# EPICS IOC start-up script: iocsh/streamMail.iocsh
################################################################################
#
# streamMail.iocsh
#
# Loads 10 user Notifiers
#
# PREFIX	- PV prefix
# MSERVER 	- mail server
# ADDRFROM  - default "source" address for user notifiers
# ADDRTO 	- default destination address for user notifiers
#
################################################################################

# set the protocol path for streamDevice
epicsEnvSet("STREAM_PROTOCOL_PATH", "$(STREAM_PROTOCOL_PATH):$(SMAIL)/sMailApp/Db")
set_requestfile_path("$(SMAIL)", "/sMailApp/Db")

drvAsynIPPortConfigure("mailPORT","$(MSERVER):25",0,0,0)

epicsEnvSet("SMPREFIX","strMail")

# Simple streamMail support
#dbLoadRecords("$(SMAIL)/sMailApp/Db/streamMail.db","P=$(PREFIX),MPORT=mailPORT,MSERVER=$(MSERVER),SM=strMail,FROM=$(ADDRFROM),TO=$(ADDRTO)")

# Load mass enable/disable
dbLoadRecords("$(SMAIL)/sMailApp/Db/streamMail_common.db","P=$(PREFIX),SM=$(SMPREFIX)")

# Load 10 notifiers
dbLoadTemplate("$(SMAIL)/sMailApp/Db/streamMail.substitutions","PREFIX=$(PREFIX),MPORT=mailPORT,MSERVER=$(MSERVER),SM=$(SMPREFIX),FROM=$(ADDRFROM),TO=$(ADDRTO)")

## Asyn record support for serial port
# use the following for troubleshooting
dbLoadRecords("$(ASYN)/db/asynRecord.db","P=$(PREFIX),R=SMasyn,PORT=mailPORT,ADDR=0,OMAX=0,IMAX=256")

#asynSetTraceIOMask("mailPORT",0,0x1)
#asynSetTraceMask("mailPORT",0,0x9)
